PROGRAM FastSignalGen
VAR
	sine	:	VariableSine;
	
	
	voltageconverter	:	ToVoltageConverter;
	
	voltageOut	AT%Q*	:	INT;
	voltageInv	AT%Q*	:	INT;
END_VAR

//sine wave generator
sine();

//sine signal to EL4132 converter
voltageconverter(in := sine.signal);
voltageOut := voltageconverter.voltage;
IF voltageOut = -32768 THEN
	voltageInv := 32767;
ELSIF voltageOut <> 0 THEN
	voltageInv := -voltageOut;
ELSE
	voltageInv := 0;
END_IF

END_PROGRAM

(* stored: Version 1.1.0.1, ProductVersion 3.1.4024.12
   POU FastSignalGen: Id {ac87b5bd-5645-4b57-bd6b-2512dc8b343d}, SpecialFunc None *)
